// TIA Portal V20 export
TYPE "typeSequenceControlNode_GRnR"
// stored: Namespace Unit1.Em9
   STRUCT
      jobs : "LAF_typeJobs";
      sequence : "LAF_typeSequence";
      selectJobStatus { S7_SetPoint := 'True'} : Array[0..10] of "LAF_typeJobStatus";
      "step" : "LER_typeStep";
      jobInterface : "Unit1.Em9.typeSequenceControlNodeJobInterface_GRnR";
   END_STRUCT;
   // // "step".action1[101] : Step[101] : JOB[1] Condition
   // // "step".action1[110] : Step[110] : Light Up
   // // "step".action1[130] : Step[130] : Stage Lift Up
   // // "step".action1[140] : Step[140] : Hot Press Right JR Detection Check
   // // "step".action1[141] : Step[141] : Hot Press Right JR Detection Check Completed
   // // "step".action1[160] : Step[160] : Stage Lift Down
   // // "step".action1[190] : Step[190] : JOB[1] Step End
   // // "step".action1[201] : Step[201] : JOB[2] Condition
   // // "step".action1[210] : Step[210] : Vision Loading Request => Transfer PP Right
   // // "step".action1[230] : Step[230] : Stage Lift Up
   // // "step".action1[240] : Step[240] : Vision Loading Check => Transfer PP Right
   // // "step".action1[290] : Step[290] : JOB[2] Step End
   // // "step".action1[301] : Step[301] : JOB[3] Condition
   // // "step".action1[310] : Step[310] : Stage Lift Down
   // // "step".action1[311] : Step[311] : Stage JR Detection Check
   // // "step".action1[320] : Step[320] : Light Down
   // // "step".action1[330] : Step[330] : Vision Start
   // // "step".action1[331] : Step[331] : Vision Result
   // // "step".action1[390] : Step[390] : JOB[3] Step End
   // // "step".action1[401] : Step[401] : JOB[4] Condition
   // // "step".action1[410] : Step[410] : Light Up
   // // "step".action1[420] : Step[420] : Stage Lift Up
   // // "step".action1[430] : Step[430] : Vision Unloading Request => Transfer PP Right
   // // "step".action1[431] : Step[431] : Vision Unloading Check => Transfer PP Right
   // // "step".action1[480] : Step[480] : Stage Lift Down
   // // "step".action1[490] : Step[490] : JOB[4] Step End
   // // "step".transition1[101] : Step[101] : JOB[1] Condition
   // // "step".transition1[110] : Step[110] : Light Up
   // // "step".transition1[130] : Step[130] : Stage Lift Up
   // // "step".transition1[140] : Step[140] : Hot Press Right JR Detection Check
   // // "step".transition1[141] : Step[141] : Hot Press Right JR Detection Check Completed
   // // "step".transition1[160] : Step[160] : Stage Lift Down
   // // "step".transition1[190] : Step[190] : JOB[1] Step End
   // // "step".transition1[201] : Step[201] : JOB[2] Condition
   // // "step".transition1[210] : Step[210] : Vision Loading Request => Transfer PP Right
   // // "step".transition1[230] : Step[230] : Stage Lift Up
   // // "step".transition1[240] : Step[240] : Vision Loading Check => Transfer PP Right
   // // "step".transition1[290] : Step[290] : JOB[2] Step End
   // // "step".transition1[301] : Step[301] : JOB[3] Condition
   // // "step".transition1[310] : Step[310] : Stage Lift Down
   // // "step".transition1[311] : Step[311] : Stage JR Detection Check
   // // "step".transition1[320] : Step[320] : Light Down
   // // "step".transition1[330] : Step[330] : Vision Start
   // // "step".transition1[331] : Step[331] : Vision Result
   // // "step".transition1[390] : Step[390] : JOB[3] Step End
   // // "step".transition1[401] : Step[401] : JOB[4] Condition
   // // "step".transition1[410] : Step[410] : Light Up
   // // "step".transition1[420] : Step[420] : Stage Lift Up
   // // "step".transition1[430] : Step[430] : Vision Unloading Request => Transfer PP Right
   // // "step".transition1[431] : Step[431] : Vision Unloading Check => Transfer PP Right
   // // "step".transition1[480] : Step[480] : Stage Lift Down
   // // "step".transition1[490] : Step[490] : JOB[4] Step End
END_TYPE
